// TIA Portal V18 export
DATA_BLOCK "DB_AI"   // DB8
{ S7_Optimized_Access := 'FALSE' }
VERSION : 0.1
// stored: AutoNumber true, DBAccessibleFromOPCUA true, DBAccessibleFromWebserver true, IsOnlyStoredInLoadMemory false, IsWriteProtectedInAS false
   VAR
      ina_InductiveResult : Real;
      ina_1 : Real;
      ina_BaseAxis : Real;
      ina_Arm1Axis : Real;
      ina_Arm2Axis : Real;
      ina_Arm3Axis : Real;
      ina_ToolAxis : Real;
      ina_7 : Real;
      ina_8 : Real;
      ina_9 : Real;
      ina_HorizontalAxis : Real;
      ina_VerticalAxis : Real;
   END_VAR
BEGIN
END_DATA_BLOCK
